
// ===== library types =====

// folder: LStream/DataTypes

TYPE "LStream_typeElement"
TITLE = LStream_typeElement
// describes the element for LStream libraries, by providing key-value pair and the depth of the element
   STRUCT
      "type" : SInt := -1;   // Type of element XML/JSON; -1 = inital value; 0 = Element/Object; 1 = Attribute/Array; 2 = Text/String; 3 = Number; 4 = Boolean / Type of element; -1 = inital value; 0 = Element/Object; 1 = Attribute/Array; 2 = Text
      key : String;   // Key name of element
      value : String := 'NULL';   // Value of element, null key has no value
      depth : SInt := -1;   // Depth of the key nesting
   END_STRUCT;
END_TYPE

// folder: LStream

FUNCTION_BLOCK "LStream_JsonDeserializer"   // FB3, SCL
TITLE = LStream_JsonDeserializer / LStream_JsonParser
{ S7_Optimized_Access := 'TRUE' }
AUTHOR : DI_FA_S_SUP_EuC
FAMILY : LStream
VERSION : 1.0
// parses a JSON string provided in the raw paramter  and rebuilds the coinatend bytes into a tree structure / Parses JSON file, with or without seach option
   VAR_INPUT
      execute : Bool;   // Rising edge starts action once
      search : Bool;   // TRUE: Search option is acticve
   END_VAR
   VAR_OUTPUT
      done : Bool;   // TRUE: Commanded functionality has been completed successfully
      busy : Bool;   // TRUE: FB is not finished and new output values can be expected
      error : Bool;   // TRUE: An error occurred during the execution of the FB
      status : Word := 16#7000;   // 16#0000 - 16#7FFF: Status of the FB, 16#8000 - 16#FFFF: Error identification
      resultCount : Int;   // Count of parsed JSON elements
   END_VAR
   VAR_IN_OUT
      tree : Array[*] of "LStream_typeElement";   // JSON tree containing the stored data
      raw : Array[*] of Byte;   // raw JSON data to parse in byte format
   END_VAR
   VAR
      statExecuteOld : Bool;   // Old value of 'execute' input for edge detection
      statDone : Bool;   // Static value for output 'done'
      statBusy : Bool;   // Static value for output 'busy'
      statError : Bool;   // Static value for output 'error'
      statStatus : Word := 16#7000;   // Static value for output 'status'
      statFBState : DInt := 0;   // State in the state machine of the FB
      statCountOfTree : Int;   // Static count of tree fields
      statCountOfRaw : Int;   // Static count of raw fields
      statResultCount : Int;   // Static value of result count
      statRawIndex : Int;   // Static value of raw index
      instWatchdog : IEC_TIMER;   // instance of watchdog timer
      statSearch : Bool;   // TRUE: Only keys provided in tree will be parsed
      statKeyValueFound : Bool;   // TRUE: Key exisits in raw data
      statTreeIndex : Int;   // Static value of tree index
      statSearchIndex : DInt;   // Static search
      statDepth : SInt := -1;   // Static value of JSON depth
      statOpen : Bool;   // TRUE: Key or Value is opened
      statInfoStartIndex : Int;   // Start index of current info in raw key or value
      statIgnorableCharacter : Bool;   // Next character to be ignored
      statInfoLen : UInt;   // Current information length key or value
      statKey : String;   // Static key string
      statValue : String;   // Static value string
      statKeyNotFoundCount : Int;   // Count of provided keys that weren't found
      statArrayOpen : Bool;   // TRUE: New JSON array is open
      statObjectArray : Bool;   // TRUE: Is type array of obejct
      statType : SInt;   // Current type of element
      statDefineValueType : Bool;   // TRUE: Value Type can be defined
      statArrayName : String;   // Name of array
   END_VAR
   VAR_TEMP
      tempExecute : Bool;   // Temporary value for input 'execute'
      tempRawIndex : Int;   // Index of raw field
      tempKeyToFind : String;   // Provided key to which the value should be found
      tempSearchResult : DInt;   // Temp value of search result
   END_VAR
   VAR CONSTANT
      FB_STATE_NO_PROCESSING : DInt := 0;   // FB state: No processing
      FB_STATE_PARSE : DInt := 1;   // FB state: Processing Parsing
      STATUS_EXECUTION_FINISHED : Word := 16#0000;   // Execution finished without errors
      STATUS_NO_CALL : Word := 16#7000;   // No job being currently processed
      STATUS_FIRST_CALL : Word := 16#7001;   // First call after incoming new job (rising edge 'execute')
      STATUS_SUBSEQUENT_CALL : Word := 16#7002;   // Subsequent call during active processing without further details
      ERR_TREE_ARRAY_TOO_SMALL : Word := 16#8201;   // Error: provided array to too small
      ERR_EMPTY_RAW_DATA : Word := 16#8401;   // Error: no raw data provided
      ERR_UNDEFINED_STATE : Word := 16#8600;   // Error: due to an undefined state in state machine
      JSON_QUTATIONMARK : Byte := 16#22;   // ASCII code for '"'
      JSON_COLON : Byte := 16#3A;   // ASCII code for ':'
      JSON_COMMA : Byte := 16#2C;   // ASCII code for ','
      JSON_BRACES_OPEN : Byte := 16#7B;   // ASCII code for '{'
      JSON_BRACES_CLOSE : Byte := 16#7D;   // ASCII code for '}'
      JSON_BRACKETS_OPEN : Byte := 16#5B;   // ASCII code for '['
      JSON_BRACKETS_CLOSE : Byte := 16#5D;   // ASCII code for ]
      "JSON_PROTECTION_KEY_\" : Byte := 16#5C;   // ASCII coder for / indicates closing / ASCII coder for \ indicates closing
      "JSON_CLOSE_KEY_/" : Byte := 16#2F;   // ASCII coder for / indicates closing
      LINE_FEED : Byte := 16#0A;   // ASCII code for line feed
      TAB : Byte := 16#09;   // ASCII code for TAB
      CARRIAGE_RETURN : Byte := 16#0D;   // ASCII code for carriage return
      SPACE : Byte := 16#20;   // ASCII code for blank space
      FIRST_DIM : USInt := 1;   // Constant for first array dimension
      MAX_LOOP_TIME : Time := T#3ms;   // Max duration of loop, will be continued in next cycle
      INVALID_SEARCH : DInt := -1;   // Return value if Search in LParse_FindStringInCharrArrayAdv was not successfull
      KEY_NOT_FOUND : String := 'Key not found';   // Value string in case key wasn't found
      INCREMENT_BY_ONE : USInt := 1;   // Constant to increment by one
      DECREMENT_BY_ONE : SInt := 1;   // Constant to decrement by one
      DECREMENT_BY_TWO : SInt := 2;   // Constant to decrement by one / Constant to decrement by two
      OBJECT : SInt := 0;   // Constant for value typ object / Constant for typ object
      "ARRAY" : SInt := 1;   // Constant for value typ array / Constant for typ array
      "STRING" : SInt := 2;   // Constant for value type string
      NUMBER : SInt := 3;   // Constant for value type number
      BOOLEAN : SInt := 4;   // Constant for value type boolean
      DEPTH_NOT_DEFINED : Int := -1;   // Constant indicating depth wasn't yet defined
   END_VAR
BEGIN
   REGION BLOCK INFO HEADER
     //===============================================================================
     // SIEMENS AG / (c)Copyright 2021
     //-------------------------------------------------------------------------------
     // Title:            LStream_JsonDeserializer
     // Comment/Function: parses a JSON string provided in the raw paramter
     //                   and rebuilds the coinatend bytes into a tree structure
     // Library/Family:   LStream
     // Author:           DI FA S SUP E&C
     // Tested with:      S7-1500 V2.8
     // Engineering:      TIA Portal V16
     // Restrictions:     -- 
     // Requirements:     LStream_FindStringInByteArrayAdv(FC), LStream_typeElement(UDT)
     //-------------------------------------------------------------------------------
     // Change log table:
     // Version  | Date       | Expert in charge       | Changes applied
     //----------|------------|------------------------|------------------------------
     // 01.0.0 | 2021-03-10 | DI FA S SUP E&C          | First released version
     // 01.0.8 | 2021-09-23 | DI FA S SUP E&C          | Adjustment type definition & bug fixes
     //===============================================================================
   END_REGION

   #tempExecute := #execute; // Work with temporary value / create process image

   REGION TRIGGERING
     IF (#tempExecute = TRUE) AND (#statExecuteOld = FALSE) // Check if FB is triggered
       AND (#statStatus = #STATUS_NO_CALL)
     THEN // First call; initialize FB
       #statDone := FALSE;
       #statBusy := TRUE;
       #statError := FALSE;
       #statStatus := #STATUS_FIRST_CALL;
       // State machine - start processing
       #statFBState := #FB_STATE_PARSE;

       // Initialize functionality: reset of variables, diagnostics, etc.
       #statSearch := #search;
       #statCountOfRaw := DINT_TO_INT(UPPER_BOUND(ARR := #raw, DIM := #FIRST_DIM));
       #statCountOfTree := DINT_TO_INT(UPPER_BOUND(ARR := #tree, DIM := #FIRST_DIM));
       #statOpen := FALSE;
       #statDepth := -1;
       #statRawIndex := 0;
       #statTreeIndex := 0;
       #statInfoLen := 0;
       #statSearchIndex := 0;
       #statKeyNotFoundCount := 0;
       #statType := -1;
       #statDefineValueType := FALSE;
       #statObjectArray := FALSE;

     ELSIF (#statStatus = #STATUS_FIRST_CALL) THEN
       #statStatus := #STATUS_SUBSEQUENT_CALL;
     END_IF;

     // Edge detection 'execute' input
     #statExecuteOld := #tempExecute;
   END_REGION TRIGGERING

   IF (#statStatus = #STATUS_NO_CALL) THEN // Nothing to do -> End here to reduce "system load"
     RETURN;
   END_IF;

   REGION STATE_MACHINE

     CASE #statFBState OF // State machine of FB
       #FB_STATE_NO_PROCESSING:
         REGION NO PROCESSING
           // No processing active (Note: this state must always be present and left empty)
           ;
         END_REGION NO PROCESSING

       #FB_STATE_PARSE: // Processing active
         REGION PARSING

           //rest watchdog
           #instWatchdog.TON(IN := FALSE,
                             PT := #MAX_LOOP_TIME);
           //start watchdog
           #instWatchdog.TON(IN := TRUE,
                             PT := #MAX_LOOP_TIME);

           FOR #tempRawIndex := #statRawIndex TO #statCountOfRaw DO

             REGION FIND KEY
               //pre check if key exist in raw data, if search option is active
               IF (#statSearch AND #statKeyValueFound = FALSE) THEN
                 IF (#statTreeIndex < #statCountOfTree) THEN
                   #tempSearchResult := "LStream_FindStringInByteCharArrayAdv"(searchFor := #tree[#statTreeIndex].key, startPosition := #statSearchIndex, searchIn := #raw);
                   IF (#tempSearchResult = #INVALID_SEARCH) THEN
                     //case key not found
                     #tree[#statTreeIndex].value := #KEY_NOT_FOUND;
                     #statTreeIndex += #INCREMENT_BY_ONE;
                     #statKeyNotFoundCount += #INCREMENT_BY_ONE;
                   ELSE//case key found
                     //move read pointer to last found index
                     #statSearchIndex := #tempSearchResult;
                     #statKeyValueFound := TRUE;
                   END_IF;
                 END_IF;
               END_IF;
             END_REGION FIND KEY   


             CASE #raw[#tempRawIndex] OF

               #JSON_BRACES_OPEN:
                 REGION OBJECT OPEN     

                   #statDepth += USINT_TO_SINT(#INCREMENT_BY_ONE);
                   IF (#statDefineValueType) THEN
                     #statDefineValueType := FALSE;
                     #statType := #OBJECT;
                     #tree[#statTreeIndex - #DECREMENT_BY_ONE].type := #statType;
                   END_IF;
                 END_REGION OBJECT OPEN

               #JSON_BRACES_CLOSE:
                 REGION OBJECT CLOSE      

                   #statDepth -= #DECREMENT_BY_ONE;
                   //last element closed, and there is still info in the buffer, then write value to last key
                   IF (#statDepth = -1 AND #statInfoLen > 0) THEN
                     //in case of 0 length, Chars_To_Strig returns the maxium possible char combination
                     Chars_TO_Strg(Chars := #raw,
                                   pChars := #statInfoStartIndex,
                                   Cnt := #statInfoLen,
                                   Strg => #statValue);
                     #statInfoLen := 0;

                     //value Type wasn't yet definied must be either number or boolean
                     IF (#statDefineValueType) THEN
                       #statDefineValueType := FALSE;

                       IF #statValue = 'FALSE' OR #statValue = 'TRUE'
                         OR #statValue = 'false' OR #statValue = 'true' THEN
                         #statType := #BOOLEAN;
                       ELSE
                         #statType := #NUMBER;
                       END_IF;

                     END_IF;

                     IF (#statSearch) THEN

                       IF (#statTreeIndex > 0) THEN
                         //in case of 0 length, Chars_To_Strig returns the maxium possible char combination
                         IF (#statKey = #tree[#statTreeIndex - #DECREMENT_BY_ONE].key) THEN
                           //only write into tree, if key matches, otherwise continue with search for matching key
                           #tree[#statTreeIndex - #DECREMENT_BY_ONE].value := #statValue;
                           #tree[#statTreeIndex - #DECREMENT_BY_ONE].type := #statType;
                           #statKeyValueFound := FALSE;
                         END_IF;
                       ELSE 
                         IF (#statKey = #tree[#statTreeIndex].key) THEN
                           #tree[#statTreeIndex].value := #statValue;
                           #tree[#statTreeIndex].type := #statType;
                           #statKeyValueFound := FALSE;
                         END_IF;
                       END_IF;

                     ELSE // IF #search option isn't active (parse all) add key TO the current #tree index
                       #tree[#statTreeIndex - #DECREMENT_BY_ONE].value := #statValue;
                       #tree[#statTreeIndex - #DECREMENT_BY_ONE].type := #statType;
                     END_IF;
                   END_IF;
                 END_REGION OBJECT CLOSE

               #JSON_BRACKETS_OPEN:
                 REGION ARRAY OPEN

                   #statDepth += USINT_TO_SINT(#INCREMENT_BY_ONE);

                   IF (#statTreeIndex > 0) THEN
                     //
                     #tree[#statTreeIndex - #DECREMENT_BY_ONE].type := #ARRAY;

                     //save arrayName
                     #statArrayName := #tree[#statTreeIndex - #DECREMENT_BY_ONE].key;

                     #statTreeIndex += #INCREMENT_BY_ONE;

                   ELSE // first element, is of type array
                     #tree[#statTreeIndex].type := #ARRAY;
                   END_IF;

                   #statArrayOpen := TRUE;
                   #statObjectArray := FALSE;
                 END_REGION ARRAY OPEN

               #JSON_BRACKETS_CLOSE:
                 REGION ARRAY CLOSE
                   #statDepth -= #DECREMENT_BY_ONE;
                   #statArrayOpen := FALSE;

                 END_REGION ARRAY CLOSE

               #JSON_QUTATIONMARK:
                 REGION QUTATIONMARK
                   IF (#statOpen) THEN
                     IF (NOT (#raw[#tempRawIndex - #DECREMENT_BY_ONE] = #"JSON_PROTECTION_KEY_\")) THEN
                       // previous sign \ then allowed in string adjust
                       #statOpen := FALSE;
                     ELSE
                       #statInfoLen += #INCREMENT_BY_ONE;
                     END_IF;
                   ELSE
                     #statInfoStartIndex := #tempRawIndex + #INCREMENT_BY_ONE; //set reader to next sign
                     #statOpen := TRUE;
                     #statIgnorableCharacter := FALSE;
                     //Qutation mark after colomn indicates value is of type string
                     IF #statDefineValueType THEN
                       #statType := #STRING;
                       #tree[#statTreeIndex - #DECREMENT_BY_ONE].type := #statType;
                       #statDefineValueType := FALSE;
                     END_IF;

                   END_IF;
                 END_REGION QUTATIONMARK

               #JSON_COLON:
                 REGION COLON

                   //array is open, and a sperate key is found indication for array of objects
                   //
                   IF #statArrayOpen AND NOT #statObjectArray THEN
                     #statObjectArray := TRUE;
                     #statTreeIndex -= #DECREMENT_BY_ONE;
                   END_IF;

                   //error handling
                   IF (#statTreeIndex > #statCountOfTree) THEN
                     //data does not fit in the provided tree 
                     #statStatus := #ERR_TREE_ARRAY_TOO_SMALL;
                     #statDone := TRUE;
                     EXIT;
                   END_IF;

                   //write key, if colon is part of a string
                   IF (NOT #statOpen) THEN
                     Chars_TO_Strg(Chars := #raw,
                                   pChars := #statInfoStartIndex,
                                   Cnt := #statInfoLen,
                                   Strg => #statKey);
                     #statInfoLen := 0;

                     //After key was written, type of value can be definied, value can be object, array, string, number, or boolean
                     #statDefineValueType := TRUE;

                     IF (#statSearch) THEN
                       //only write into tree, if key matches, otherwise continue with search for matching key
                       IF (#statKey = #tree[#statTreeIndex].key) THEN
                         //#tree[#statTreeIndex].type := #statType;
                         #tree[#statTreeIndex].depth := #statDepth;
                         #statTreeIndex += #INCREMENT_BY_ONE;
                       END_IF;

                     ELSE// if search option isn't active (parse all) the add key to the current tree index 
                       #tree[#statTreeIndex].key := #statKey;
                       //#tree[#statTreeIndex].type := #statType;
                       #tree[#statTreeIndex].depth := #statDepth;
                       #tree[#statTreeIndex].value := 'NULL';
                       #statTreeIndex += #INCREMENT_BY_ONE;
                     END_IF;

                     #statInfoStartIndex := #tempRawIndex+1;

                   ELSE//case : included in string
                     #statInfoLen += #INCREMENT_BY_ONE;
                   END_IF;
                 END_REGION COLON

               #JSON_COMMA:
                 REGION COMMA

                   //error handling
                   IF (#statTreeIndex > #statCountOfTree + #INCREMENT_BY_ONE) THEN
                     //data does not fit in the provided tree 
                     #statStatus := #ERR_TREE_ARRAY_TOO_SMALL;
                     #statDone := TRUE;
                     EXIT;
                   END_IF;

                   IF (NOT #statOpen) THEN
                     //write value comma isn't part of string
                     IF (#statInfoLen > 0) THEN
                       //in case of 0 length, Chars_To_Strig returns the maxium possible char combination
                       Chars_TO_Strg(Chars := #raw,
                                     pChars := #statInfoStartIndex,
                                     Cnt := #statInfoLen,
                                     Strg => #statValue);
                       #statInfoLen := 0;
                     ELSE
                       #statValue := 'NULL';
                       #statDefineValueType := FALSE;
                       //no value Type deafult value type NULL/Default is correct
                     END_IF;

                     //value Type wasn't yet definied must be either number or boolean
                     IF (#statDefineValueType) THEN
                       #statDefineValueType := FALSE;

                       IF #statValue = 'FALSE' OR #statValue = 'TRUE'
                         OR #statValue = 'false' OR #statValue = 'true' THEN
                         #statType := #BOOLEAN;
                       ELSE
                         #statType := #NUMBER;
                       END_IF;

                     END_IF;
                     //add value always to the last JSON element
                     IF (#statSearch) THEN

                       IF (#statTreeIndex > 0) THEN
                         //in case of 0 length, Chars_To_Strig returns the maxium possible char combination
                         IF (#statKey = #tree[#statTreeIndex - #DECREMENT_BY_ONE].key) THEN
                           //only write into tree, if key matches, otherwise continue with search for matching key
                           #tree[#statTreeIndex - #DECREMENT_BY_ONE].value := #statValue;
                           #tree[#statTreeIndex].type := #statType;
                           #statKeyValueFound := FALSE;
                         END_IF;
                       ELSE
                         IF (#statKey = #tree[#statTreeIndex].key) THEN
                           // if search option isn't active (parse all) the add key to the current tree index 
                           #tree[#statTreeIndex].value := #statValue;
                           #tree[#statTreeIndex].type := #statType;
                           #statKeyValueFound := FALSE;
                         END_IF;
                       END_IF;

                     ELSE//search option isn't active
                       #tree[#statTreeIndex - #DECREMENT_BY_ONE].value := #statValue;
                       #tree[#statTreeIndex - #DECREMENT_BY_ONE].type := #statType;
                       //case simple array last information
                       IF (#tree[#statTreeIndex - #DECREMENT_BY_ONE].depth = #DEPTH_NOT_DEFINED) THEN
                         #tree[#statTreeIndex - #DECREMENT_BY_ONE].depth := #tree[#statTreeIndex - #DECREMENT_BY_TWO].depth;
                         #tree[#statTreeIndex - #DECREMENT_BY_ONE].key := #statArrayName;
                         //always take depth from previous entry of simple array e.g "ArrayName":["ArrayValue1","ArrayValue2"]
                       END_IF;
                     END_IF;

                     IF (#statArrayOpen AND NOT #statObjectArray) THEN
                       //only write if Array is open and simple array
                       //
                       #tree[#statTreeIndex- #DECREMENT_BY_ONE].key := #statArrayName;
                       #tree[#statTreeIndex - #DECREMENT_BY_ONE].depth := #statDepth;//#tree[#statTreeIndex - #DECREMENT_BY_TWO].depth +1;
                       #tree[#statTreeIndex- #DECREMENT_BY_ONE].type := #statType;
                       //always take depth from previous entry of simple array e.g "ArrayName":["ArrayValue1","ArrayValue2"]


                       // #tree[#statTreeIndex].key := #tree[#statTreeIndex - #DECREMENT_BY_ONE].key;
                       // #tree[#statTreeIndex].depth := #tree[#statTreeIndex - #DECREMENT_BY_ONE].depth;
                       // #tree[#statTreeIndex].type := #tree[#statTreeIndex - #DECREMENT_BY_ONE].type;
                       #statTreeIndex += #INCREMENT_BY_ONE;
                     END_IF;

                     #statInfoStartIndex := #tempRawIndex;

                   ELSE//case ; included in string
                     #statInfoLen += #INCREMENT_BY_ONE;
                   END_IF;
                 END_REGION

               #TAB, #LINE_FEED, #CARRIAGE_RETURN, #SPACE:
                 REGION READ TAB LINE FEED CARRIAGE RETURN   
                   IF (NOT #statOpen) THEN
                     //do nothing when tab, line feed, or carriage return
                     #statIgnorableCharacter := TRUE;
                   ELSE//case space included in string
                     #statInfoLen += #INCREMENT_BY_ONE;
                   END_IF;

                 END_REGION READ TAB LINE FEED CARRIAGE RETURN     


               ELSE // all other characters
                 REGION ALL OTHER SIGNS
                 IF (#statIgnorableCharacter = TRUE) THEN
                   #statIgnorableCharacter := FALSE;
                   #statInfoStartIndex := #tempRawIndex; // set KeyIndex after all ignorableCharacters are read
                   #statInfoLen += #INCREMENT_BY_ONE;
                 ELSE
                   #statInfoLen += #INCREMENT_BY_ONE;
                 END_IF;
                 END_REGION ALL OTHER SIGNS 
             END_CASE;

             #statRawIndex := #tempRawIndex;

             //quit and resume in next cycle if watchdogtimer is exceed
             IF (#instWatchdog.Q) THEN
               #statRawIndex += #INCREMENT_BY_ONE;
               EXIT;
             END_IF;

           END_FOR;

           //if parser is through the entire raw data or end of tree array reached
           IF (#statRawIndex >= #statCountOfRaw) OR (#statTreeIndex > #statCountOfTree) THEN
             #statStatus := #STATUS_EXECUTION_FINISHED;
             #statResultCount := #statTreeIndex - #statKeyNotFoundCount;
           END_IF;
         END_REGION PARSING

       ELSE // Undefined state in state machine reached
         REGION UNDEFINED STATE
           #statStatus := #ERR_UNDEFINED_STATE;
         END_REGION UNDEFINED STATE
     END_CASE;
   END_REGION STATE_MACHINE

   REGION OUTPUTS
     // Write outputs
     IF (#statStatus = #STATUS_EXECUTION_FINISHED) AND (#statDone = FALSE) THEN // Execution finished without errors
       REGION EXECUTION FINSIHED
         #statDone := TRUE;
         #statBusy := FALSE;
         #statError := FALSE;
         // execution aborted --> set state no processing
         #statFBState := #FB_STATE_NO_PROCESSING;
       END_REGION EXECUTION FINSIHED

     ELSIF (#statStatus.%X15 = TRUE) AND (#statError = FALSE) THEN // Error occurred (#statStatus is 16#8000 to 16#FFFF)
       REGION ERROR OCCURD
         #statDone := FALSE;
         #statBusy := FALSE;
         #statError := TRUE;
         // execution aborted --> set state no processing
         #statFBState := #FB_STATE_NO_PROCESSING;
       END_REGION ERROR OCCURD

     ELSIF (#tempExecute = FALSE) AND ((#statDone = TRUE) OR (#statError = TRUE)) THEN // Reset outputs
       REGION EXECUTE RESETED
         #statDone := FALSE;
         #statBusy := FALSE;
         #statError := FALSE;
         #statStatus := #STATUS_NO_CALL;
         // Reset application specific outputs
         #statResultCount := 0;
       END_REGION EXECUTE RESETED
     END_IF;

     REGION WRITE STATIC VALUES TO OUTPUTS
       #done := #statDone;
       #busy := #statBusy;
       #error := #statError;
       #status := #statStatus;

       ENO := TRUE;
       // Write application specific static values to outputs
       #resultCount := #statResultCount;
     END_REGION WRITE STATIC VALUES TO OUTPUT
   END_REGION OUTPUTS
END_FUNCTION_BLOCK

FUNCTION_BLOCK "LStream_XmlDeserializer"   // FB4, SCL
TITLE = LStream_XmlDeserializer / LStream_Xml
{ S7_Optimized_Access := 'TRUE' }
AUTHOR : DI_FA_S_SUP_EuC
FAMILY : LStream
VERSION : 1.0
// parses a XML string provided in the Raw parameter and rebuilds the contained tree structure / Function Block parses entire or partial XML into DB
   VAR_INPUT
      execute : Bool;   // Rising edge starts action once
      search : Bool;   // TRUE: Searches rawdata for the value of the provided treekeys
   END_VAR
   VAR_OUTPUT
      done : Bool;   // TRUE: Commanded functionality has been completed successfully
      busy : Bool;   // TRUE: FB is not finished and new output values can be expected
      error : Bool;   // TRUE: An error occurred during the execution of the FB
      status : Word := 16#7000;   // 16#0000 - 16#7FFF: Status of the FB, 16#8000 - 16#FFFF: Error identification
      resultCount : Int;   // Count of parsed XML elements
   END_VAR
   VAR_IN_OUT
      tree : Array[*] of "LStream_typeElement";   // Tree parsed information is written to, if search option active, keys must be provided
      raw : Array[*] of Byte;   // Byte array of raw xml data
   END_VAR
   VAR
      statOldExecute : Bool;   // Old value of 'execute' input for edge detection
      statDepth : SInt := -1;   // Static value of xml depth
      statError : Bool;   // Static value of error
      statBusy : Bool;   // Static value of busy
      statStatus : Word := 16#7000;   // Static value of status
      statFBState : USInt := 0;   // Static value of fb state
      statDone : Bool;   // Static value of done
      statResultCount : Int;   // Static value of result count
      instWatchdog : IEC_TIMER;   // Instance of watchdog timer
      statRawIndex : Int;   // Static value of raw index
      statTreeIndex : Int;   // Static value of tree index
      statCountOfTree : Int;   // Static count of tree fields
      statCountOfRaw : Int;   // Static count of raw fields
      statIsIgnorable : Bool;   // Ignore any sign
      statIsKeyOpen : Bool;   // TRUE: key is open, internal flag
      statIsValueOpen : Bool;   // TRUE: value is open, internal flag
      statInfoLen : UInt;   // Current information length key or value
      statLastElementTreeIndex : Int;   // Treeindex of last element found
      statIgnorableCharacter : Bool;   // Next character to be ignored
      statInfoStartIndex : Int;   // Start index of current info in raw key or value
      statKeyWritten : Bool;   // TRUE: key was written into tree
      statKey : String;   // Static key string
      statValue : String;   // Static value string
      statSearch : Bool;   // TRUE: Only keys provided in tree will be parsed
      statKeyFound : Bool;   // TRUE: Key exisits in raw data
      statKeyNotFoundCount : Int;   // Count of provided keys that weren't found
      statSearchIndex : DInt;   // Static search index
   END_VAR
   VAR_TEMP
      tempRawIndex : Int;   // Index of raw field
      tempExecute : Bool;   // Temp of input execute
      tempKeyToFind : String;   // Provided key to which the value should be found
      tempSearchResult : DInt;   // Temp value of search result
   END_VAR
   VAR CONSTANT
      INCREMENT_BY_ONE : SInt := 1;   // Constant to increment by one
      DECREMENT_BY_ONE : SInt := 1;   // Constant to decrement by one
      FB_STATE_NO_PROCESSING : USInt := 0;   // FB state no processing, ideal state
      FB_STATE_PARSE : USInt := 10;   // FB state parse xml
      FB_STATE_DONE : USInt := 70;   // FB state done
      STATUS_EXECUTION_FINISHED : Word := 16#0000;   // NO error - execution finished without errors
      STATUS_NO_CALL : Word := 16#7000;   // No job being currently processed
      STATUS_FIRST_CALL : Word := 16#7001;   // First call after incoming new job (rising edge 'execute')
      STATUS_SUBSEQUENT_CALL : Word := 16#7002;   // Subsequent call during active processing without further details
      ERR_TREE_ARRAY_TOO_SMALL : Word := 16#8201;   // Error: provided array to too small
      ERR_EMPTY_RAW_DATA : Word := 16#8401;   // Error: no raw data provided
      ERR_UNDEFINED_STATE : Word := 16#8600;   // Error: due to an undefined state in state machine
      XML_HEADER : Byte := 16#3F;   // ASCII code for ? indicates xml header
      XML_COMMENT : Byte := 16#21;   // ASCII code for ! indicates comment
      XML_ATTRIBUTE_OPEN : Byte := 16#22;   // ASCII code for " frames value
      XML_OPEN_KEY : Byte := 16#3C;   // ASCII code for < indicates a new key
      XML_WRITE_KEY_EQUALS : Byte := 16#3D;   // ASCII code for '=' indicates key is finished follows by value
      XML_WRITE_KEY_GREATER : Byte := 16#3E;   // ASCII code for > indicates key can be written
      XML_WRITE_KEY_SPACE : Byte := 16#20;   // ASCII codefor SPACE indicates key is finished
      XML_CLOSE_KEY_SLASH : Byte := 16#2F;   // ASCII code for / indicates closing
      CARRIAGE_RETURN : Byte := 16#0D;   // ASCII code for carriage return
      LINE_FEED : Byte := 16#0A;   // ASCII code for line feed
      TAB : Byte := 16#09;   // ASCII code for TAB
      EMPTY : SInt := 0;   // Constant for zero value
      ELEMENT : SInt := 0;   // Numerical identifier for XML type elemt
      ATTRIBUTE : SInt := 1;   // Numerical identifier for XML type attirbute
      TEXT : SInt := 2;   // Numerical identifier for XML type text
      FIRST_DIM : USInt := 1;   // Constant for first array dimension
      MAX_LOOP_TIME : Time := T#3ms;   // Max duration of loop, will be continued in next cycle
      INVALID_SEARCH : DInt := -1;   // Return value if Search in LParse_FindStringInCharrArrayAdv was not successfull
      KEY_NOT_FOUND : String := 'Key not found';   // String value in case key wasn't found
   END_VAR
BEGIN
   REGION BLOCK INFO HEADER
     //===============================================================================
     // SIEMENS AG / (c)Copyright 2021
     //-------------------------------------------------------------------------------
     // Title:            LStream_XmlDeserializer
     // Comment/Function: parses a XML string provided in the Raw parameter
     //                   and rebuilds the contained tree structure
     // Library/Family:   LStream
     // Author:           DI FA S SUP E&C
     // Tested with:      S7-1500 V2.8
     // Engineering:      TIA Portal V16
     // Restrictions:     --
     // Requirements:     LStream_FindStringInByteArrayAdv(FC), LStream_typeElement(UDT)
     //-------------------------------------------------------------------------------
     // Change log table:
     // Version  | Date       | Expert in charge | Changes applied
     //----------|------------|------------------|------------------------------------
     // 01.00.00 | 2021-03-10 | DI FA S SUP E&C  | First released version
     //===============================================================================
   END_REGION

   #tempExecute := #execute;

   REGION TRIGGERING 

     IF (#tempExecute = TRUE) AND (#statOldExecute = FALSE)
       AND (#statStatus = #STATUS_NO_CALL)
     THEN // First call; initialize FB

       #statDone := FALSE;
       #statBusy := TRUE;
       #statStatus := #STATUS_FIRST_CALL;

       // Initialize functionality: reset of variables, diagnostics, etc.
       #statSearch := #search;
       #statCountOfRaw := DINT_TO_INT(UPPER_BOUND(ARR := #raw, DIM := #FIRST_DIM));
       #statCountOfTree := DINT_TO_INT(UPPER_BOUND(ARR := #tree, DIM := #FIRST_DIM));
       #statDepth := 0;
       #statRawIndex := 0;
       #statTreeIndex := 0;
       #statIsIgnorable := FALSE;
       #statIsKeyOpen := FALSE;
       #statIsValueOpen := FALSE;
       #statKeyWritten := FALSE;
       #statInfoLen := 0;
       #statLastElementTreeIndex := 0;
       #statIgnorableCharacter := FALSE;
       #statInfoStartIndex := 0;
       #statKey := '';
       #statValue := '';
       #statKeyFound := FALSE;
       #statSearchIndex := 0;
       #statKeyNotFoundCount := 0;

       // State machine - start processing
       #statFBState := #FB_STATE_PARSE;

       IF (NOT (#statCountOfRaw > #EMPTY)) THEN
         #statStatus := #ERR_EMPTY_RAW_DATA;
       END_IF;

     ELSIF (#statStatus = #STATUS_FIRST_CALL) THEN
       #statStatus := #STATUS_SUBSEQUENT_CALL;

     END_IF;

     // Edge detection 'execute' input
     #statOldExecute := #tempExecute;
   END_REGION TRIGGERING 

   IF (#statStatus = #STATUS_NO_CALL) THEN // Nothing to do -> End here to reduce "system load"
     RETURN;
   END_IF;

   REGION PROGRAM LOGIC

     CASE #statFBState OF // State machine of FB

       #FB_STATE_NO_PROCESSING:
         REGION NO PROCESSING
           // No processing active (Note: this state must always be present AND left empty)
           ;
         END_REGION NO PROCESSING           

       #FB_STATE_PARSE:
         REGION PARSE XML

           //rest and start watchdog here so that for loop runs for a maximum of 5 seconds
           #instWatchdog.TON(IN := FALSE,
                             PT := #MAX_LOOP_TIME);
           //start watchdog
           #instWatchdog.TON(IN := TRUE,
                             PT := #MAX_LOOP_TIME);

           FOR #tempRawIndex := #statRawIndex TO #statCountOfRaw DO

             //pre check if key exist in raw data, only if search option is active and key wasn't already found
             IF (#statSearch AND #statKeyFound = FALSE) THEN
               IF (#statTreeIndex < #statCountOfTree) THEN
                 #tempSearchResult := "LStream_FindStringInByteCharArrayAdv"(searchFor := #tree[#statTreeIndex].key, startPosition := #statSearchIndex, searchIn := #raw);

                 IF (#tempSearchResult = #INVALID_SEARCH) THEN
                   //case key not found
                   #tree[#statTreeIndex].value := #KEY_NOT_FOUND;
                   #statTreeIndex += #INCREMENT_BY_ONE;
                   #statKeyNotFoundCount += #INCREMENT_BY_ONE;

                 ELSE //case key found
                   //move read pointer to last found index
                   #statSearchIndex := #tempSearchResult;
                   #statKeyFound := TRUE;
                 END_IF;
               END_IF;
             END_IF;

             //swich case of current byte
             CASE #raw[#tempRawIndex] OF

               #XML_OPEN_KEY:
                 REGION READ OPENING KEY SYMBOLS                            
                   //check if is XML Header or comment by looking ahead by one 
                   IF (#raw[#tempRawIndex + 1] = #XML_HEADER) OR (#raw[#tempRawIndex + 1] = #XML_COMMENT) THEN
                     //in xml case <? and <!, ignore all signs until header or comment is finished
                     #statIsIgnorable := true;
                     #statInfoLen := 0;
                     //rest length buffer

                     //look ahead for closing  
                   ELSIF (#raw[#tempRawIndex + 1] = #XML_CLOSE_KEY_SLASH) THEN
                     // xml case </ indicates closeing
                     #statIsKeyOpen := false;
                     #statInfoLen := 0;

                   ELSE //indicates opening 
                     IF (#statTreeIndex > #statCountOfTree + #INCREMENT_BY_ONE) THEN
                       //data does not fit in the provided tree
                       #statStatus := #ERR_TREE_ARRAY_TOO_SMALL;
                       #statDone := TRUE;
                       EXIT;
                     END_IF;

                     IF (#statInfoLen > #EMPTY AND #statIsKeyOpen = TRUE) THEN
                       //xml case >text< 

                       Chars_TO_Strg(Chars := #raw,
                                     pChars := #statInfoStartIndex,
                                     Cnt := #statInfoLen,
                                     Strg => #statValue);

                       //add value to the last xml element
                       IF (#statSearch) THEN // search option is active

                         //only write value into tree, if key matches, otherwise continue with search for matching key
                         IF (#statKey = #tree[#statTreeIndex - #DECREMENT_BY_ONE].key) THEN

                           #tree[#statTreeIndex - #DECREMENT_BY_ONE].depth := #statDepth;
                           #tree[#statTreeIndex - #DECREMENT_BY_ONE].value := #statValue;
                           #tree[#statTreeIndex - #DECREMENT_BY_ONE].type := #TEXT;

                         END_IF;

                       ELSE // if search option isn't active (parse all) the value must be attached to the last key
                         #tree[#statTreeIndex - #DECREMENT_BY_ONE].depth := #statDepth;
                         #tree[#statTreeIndex - #DECREMENT_BY_ONE].value := #statValue;
                         #tree[#statTreeIndex - #DECREMENT_BY_ONE].type := #TEXT;
                       END_IF;
                     END_IF;

                     // new element
                     #statKeyWritten := FALSE;
                     #statIsKeyOpen := TRUE;
                     #statDepth += #INCREMENT_BY_ONE;
                     #statInfoStartIndex := #tempRawIndex + #INCREMENT_BY_ONE;
                     #statInfoLen := 0;

                   END_IF;

                 END_REGION READ OPENING KEY SYMBOLS       

               #XML_WRITE_KEY_GREATER, #XML_WRITE_KEY_EQUALS, #XML_WRITE_KEY_SPACE:
                 REGION READ WRITING KEY SYMBOLS

                   IF (#statIsIgnorable = FALSE) THEN
                     IF (#statInfoLen > #EMPTY AND #statIsKeyOpen = TRUE) THEN

                       IF (#statTreeIndex > #statCountOfTree) THEN
                         //data does not fit in the provided tree
                         #statStatus := #ERR_TREE_ARRAY_TOO_SMALL;
                         #statDone := TRUE;
                         EXIT;
                       END_IF;

                       Chars_TO_Strg(Chars := #raw,
                                     pChars := #statInfoStartIndex,
                                     Cnt := #statInfoLen,
                                     Strg => #statKey);


                       IF (#statSearch) THEN
                         //only write into tree, if key matches, otherwise continue with search for matching key
                         IF (#statKey = #tree[#statTreeIndex].key) THEN
                           #tree[#statTreeIndex].depth := #statDepth;
                           #tree[#statTreeIndex].type := #ELEMENT;
                           #statTreeIndex += #INCREMENT_BY_ONE;
                           #statKeyFound := FALSE;
                         END_IF;

                       ELSE// if search option isn't active (parse all) the add key to the current tree index
                         #tree[#statTreeIndex].key := #statKey;
                         #tree[#statTreeIndex].type := #ELEMENT;
                         #tree[#statTreeIndex].depth := #statDepth;
                         #tree[#statTreeIndex].value := 'NULL';
                         #statLastElementTreeIndex := #statTreeIndex;
                         #statTreeIndex += #INCREMENT_BY_ONE;
                         #statKeyFound := FALSE;
                         #statKeyWritten := TRUE;

                       END_IF;

                       #statInfoLen := 0;

                     END_IF;

                     #statInfoStartIndex := #tempRawIndex + #INCREMENT_BY_ONE;

                   ELSIF (#statIsIgnorable = TRUE AND #raw[#tempRawIndex] = #XML_WRITE_KEY_GREATER) THEN
                     //xml case closing of <? and <!, stop ignoring all signs
                     //only if sign is >
                     #statIsIgnorable := FALSE;

                   END_IF;
                 END_REGION READ WRITING KEY SYMBOLS

               #XML_CLOSE_KEY_SLASH:
                 REGION READ DELIMETER /
                   #statDepth -= #DECREMENT_BY_ONE;
                   #statIsKeyOpen := false;

                   IF (#statTreeIndex > #statCountOfTree) THEN
                     //data does not fit in the provided tree
                     #statStatus := #ERR_TREE_ARRAY_TOO_SMALL;
                     #statDone := TRUE;
                     EXIT;
                   END_IF;

                   IF (#statKeyWritten = FALSE) THEN
                     Chars_TO_Strg(Chars := #raw,
                                   pChars := #statInfoStartIndex,
                                   Cnt := #statInfoLen,
                                   Strg => #statKey);

                     //only if key wasn't alrady written
                     IF (NOT (#tree[#statLastElementTreeIndex].key = #statKey)) THEN

                       IF (#statSearch) THEN
                         //only write into tree, if key matches, otherwise continue with search for matching key
                         IF (#statKey = #tree[#statTreeIndex].key) THEN
                           #tree[#statTreeIndex].depth := #statDepth;
                           #statLastElementTreeIndex := #statTreeIndex;
                           #statTreeIndex += #INCREMENT_BY_ONE;
                           #statKeyFound := FALSE;
                         END_IF;
                       ELSE
                         // if search option isn't active (parse all) the add key to the current tree index
                         #tree[#statTreeIndex].key := #statKey;
                         #tree[#statTreeIndex].type := #ELEMENT;
                         #tree[#statTreeIndex].depth := #statDepth;
                         #tree[#statTreeIndex].value := 'NULL';
                         #statLastElementTreeIndex := #statTreeIndex;
                         #statTreeIndex += #INCREMENT_BY_ONE;
                         #statKeyFound := FALSE;
                         #statKeyWritten := TRUE;
                         #statInfoStartIndex := #tempRawIndex + #INCREMENT_BY_ONE;
                       END_IF;
                     END_IF;

                     #statInfoLen := 0;
                   END_IF;

                 END_REGION READ DELIMETER /

               #XML_ATTRIBUTE_OPEN:
                 REGION READ VALUE SYMBOLES
                   IF (#statIsIgnorable = FALSE) THEN

                     IF (#statIsValueOpen = false) THEN //first enter indicates begin of value
                       #statIsValueOpen := true;
                       #statInfoStartIndex := #tempRawIndex + #INCREMENT_BY_ONE;

                     ELSE // second enter indicates end of value
                       #statIsValueOpen := false;

                       IF (#statTreeIndex > #statCountOfTree + #INCREMENT_BY_ONE) THEN
                         //data does not fit in the provided tree 
                         #statStatus := #ERR_TREE_ARRAY_TOO_SMALL;
                         #statDone := TRUE;
                         EXIT;
                       END_IF;

                       //attach value to last key node
                       Chars_TO_Strg(Chars := #raw,
                                     pChars := #statInfoStartIndex,
                                     Cnt := #statInfoLen,
                                     Strg => #statValue);

                       IF (#statSearch) THEN
                         //only write into tree, if key matches, otherwise continue with search for matching key
                         IF (#statKey = #tree[#statTreeIndex - #DECREMENT_BY_ONE].key) THEN
                           #tree[#statTreeIndex - #DECREMENT_BY_ONE].depth := #statDepth;
                           #tree[#statTreeIndex - #DECREMENT_BY_ONE].value := #statValue;
                           #tree[#statTreeIndex - #DECREMENT_BY_ONE].type := #ATTRIBUTE;

                         END_IF;
                       ELSE
                         // if search option isn't active (parse all) the add key to the current tree index
                         #tree[#statTreeIndex - #DECREMENT_BY_ONE].value := #statValue;
                         #tree[#statTreeIndex - #DECREMENT_BY_ONE].type := #ATTRIBUTE;
                         #tree[#statTreeIndex - #DECREMENT_BY_ONE].depth := #statDepth;

                         #statIsValueOpen := false;
                       END_IF;
                       #statInfoLen := 0;
                     END_IF;
                   END_IF;
                 END_REGION READ VALUE SYMBOLES     

               #TAB, #LINE_FEED, #CARRIAGE_RETURN:
                 REGION READ TAB LINE FEED CARRIAGE RETURN                      
                   #statIgnorableCharacter := TRUE;
                   //do nothing when tab, line feed, or carriage return
                 END_REGION READ TAB LINE FEED CARRIAGE RETURN

               ELSE//all other characters  
                 REGION READ OTHER SIGN
                   IF (#statIgnorableCharacter = TRUE) THEN
                     #statIgnorableCharacter := FALSE;
                     #statInfoStartIndex := #tempRawIndex; // set KeyIndex after all ignorableCharacters are read

                   END_IF;
                   //count length in case not header or comment
                   IF (#statIsIgnorable = FALSE) THEN
                     #statInfoLen += SINT_TO_UINT(#INCREMENT_BY_ONE);
                   END_IF;

                 END_REGION READ OTHER SIGN                         

             END_CASE;
             #statRawIndex := #tempRawIndex;

             //quit and resume in next cycle if watchdogtimer is exceed
             IF (#instWatchdog.Q) THEN
               #statRawIndex += #INCREMENT_BY_ONE;
               EXIT;
             END_IF;
           END_FOR;

           //if parser is through the entire raw data or end of tree array reached
           IF (#statRawIndex >= #statCountOfRaw) OR (#statTreeIndex > #statCountOfTree) THEN
             #statStatus := #STATUS_EXECUTION_FINISHED;
             #statResultCount := #statTreeIndex - #statKeyNotFoundCount;
           END_IF;
         END_REGION PARSE XML              

       ELSE // Undefined state in state machine reached
         REGION UNDEFINED STATE
           #statStatus := #ERR_UNDEFINED_STATE;
         END_REGION UNDEFINED STATE
     END_CASE;

   END_REGION PROGRAM LOGIC

   REGION OUTPUTS

     // Write outputs
     IF (#statStatus = #STATUS_EXECUTION_FINISHED) AND (#statDone = FALSE) THEN // Execution finished without errors
       REGION EXECUTION FINISHED
         #statDone := TRUE;
         #statBusy := FALSE;
         #statError := FALSE;
         // execution aborted --> set state no processing
         #statFBState := #FB_STATE_NO_PROCESSING;
       END_REGION EXECUTION FINISHED

     ELSIF (#statStatus.%X15 = TRUE) AND (#statError = FALSE) THEN // Error occurred (#statStatus is 16#8000 to 16#FFFF)
       REGION ERROR OCCURED
         #statDone := FALSE;
         #statBusy := FALSE;
         #statError := TRUE;
         // execution aborted --> set state no processing
         #statFBState := #FB_STATE_NO_PROCESSING;
       END_REGION ERROR OCCURED

     ELSIF (#tempExecute = FALSE) AND ((#statDone = TRUE) OR (#statError = TRUE)) THEN // Reset outputs
       REGION EXECUTE RESETED
         #statDone := FALSE;
         #statBusy := FALSE;
         #statError := FALSE;
         #statStatus := #STATUS_NO_CALL;
         // Reset application specific outputs
         #statResultCount := 0;
       END_REGION EXECUTE RESETED
     END_IF;

     REGION WRITE STATIC VALUES TO OUTPUTS
       // write application specific temp values to outputs
       #resultCount := #statResultCount;
       #done := #statDone;
       #error := #statStatus.%X15;
       #status := #statStatus;
       #busy := #statBusy;

     END_REGION WRITE STATIC VALUES TO OUTPUTS

   END_REGION OUTPUTS
END_FUNCTION_BLOCK

FUNCTION_BLOCK "LStream_JsonSerializer"   // FB5, SCL
TITLE = LStream_JsonDeserializer / LStream_JsonParser
{ S7_Optimized_Access := 'TRUE' }
AUTHOR : DI_FA_S_SUP_EuC
FAMILY : LStream
VERSION : 1.0
// parses a JSON string provided in the raw paramter  and rebuilds the coinatend bytes into a tree structure / Parses JSON file, with or without seach option
   VAR_INPUT
      execute : Bool;   // Rising edge starts action once
   END_VAR
   VAR_OUTPUT
      done : Bool;   // TRUE: Commanded functionality has been completed successfully
      busy : Bool;   // TRUE: FB is not finished and new output values can be expected
      error : Bool;   // TRUE: An error occurred during the execution of the FB
      status : Word := 16#7000;   // 16#0000 - 16#7FFF: Status of the FB, 16#8000 - 16#FFFF: Error identification
      count : UInt;   // Count of char/ byte info elements in byte array / Count of parsed JSON elements
   END_VAR
   VAR_IN_OUT
      tree : Array[*] of "LStream_typeElement";   // JSON tree containing the stored data
      jsonByteArray : Array[*] of Byte;   // JSON structure as array of bytes / raw JSON data to parse in byte format
   END_VAR
   VAR
      statExecuteOld : Bool := FALSE;   // Old value of 'execute' input for edge detection
      statDone : Bool := FALSE;   // Static value for output 'done'
      statBusy : Bool := FALSE;   // Static value for output 'busy'
      statError : Bool := FALSE;   // Static value for output 'error'
      statCount : UInt := 0;   // Static value for ouput 'count'
      statStatus : Word := 16#7000;   // Static value for output 'status'
      statFbState : DInt := 0;   // State in the state machine of the FB
      statFbPreviousState : DInt := 0;   // Previos state in the state machine of the FB
      statFbNextState : DInt := 0;   // Next state in the state machine of the FB
      statIndexJsonByteArray : UInt := 0;   // Index indicating current element of byte array to be written
      statIndexTreeArray : UInt := 0;   // Index indicating current element of tree array to be read
      statTreeLen : DInt := 0;   // Length of tree array
      statJsonByteLen : DInt := 0;   // Length of xml byte array / Length of json byte array
      statInfoToWrite : String := '';   // Static value of current information that should be written to XML
      statIsLastElement : Bool := FALSE;   // TRUE: is last element in tree array
      statLastElementIsClosed : Bool := FALSE;   // TRUE: Last JSON element is closed / TRUE: Last XML element is closed
      statStackIndexOpenElement : Array[0..#STACK_SIZE] of Char;   // Stack of open elements
      statStackIndex : Int := -1;   // Stack pointer and current depth / Stack pointer
      instWatchdog : IEC_TIMER;   // Instance for watchdog timer
      statIsArrayOpen : Bool;   // Static value indicating weather an array is open
      statIsArrayFieldClosed : Bool;   // Static value indicating weather an array field was closed
      statIsFirstElement : Bool;   // TRUE: first field of simple array
      statFirstArrayKey : String;   // First key of array, used to check for new array beginning
      statArrayName : String;   // Name of Array
   END_VAR
   VAR_TEMP
      tempExecute : Bool;   // Temporary value for input 'execute'
      tempCntCharsAdded : UInt;   // Temporary value indicating count of chars added to byte array
   END_VAR
   VAR CONSTANT
      FB_STATE_NO_PROCESSING : DInt := 0;   // FB state: No processing
      FB_STATE_NEXT_ELEMENT : DInt := 1;   // FB state: Get Next Element
      FB_STATE_VALUE_TYPE : DInt := 2;   // FB state: Switch Value type / FB state: Switch Element type
      FB_STATE_WRITE_TO_JSON : DInt := 3;   // FB state: Add Informationto xml byte array
      FB_STATE_CLOSE_STACK_ELEMENT : DInt := 4;   // FB state: Close Parent Element
      STATUS_EXECUTION_FINISHED : Word := 16#0000;   // Execution finished without errors
      STATUS_NO_CALL : Word := 16#7000;   // No job being currently processed
      STATUS_FIRST_CALL : Word := 16#7001;   // First call after incoming new job (rising edge 'execute')
      STATUS_SUBSEQUENT_CALL : Word := 16#7002;   // Subsequent call during active processing without further details
      ERR_UNDEFINED_STATE : Word := 16#8600;   // Error: due to an undefined state in state machine
      ERR_IN_BLOCK_OPERATION : Word := 16#8001;   // Error: wrong operation of the function block
      ERR_PARAMETRIZATION : Word := 16#8200;   // Error: during parameterization
      ERR_PROCESSING_EXTERN : Word := 16#8400;   // Error: when processing from outside (e. g. wrong I/O signals, axis not referenced)
      ERR_UNDEFINED_TYPE : Word := 16#8401;   // Error: user enter undefined type
      ERR_UNEXPECTED_DEPTH : Word := 16#8402;   // Error: provided json tree structure is too deep / Error: provided xml tree structure is too deep
      ERR_DEPTH_MISSING : Word := 16#8403;   // Error: provided json tree structure does not contain correct depth / Error: provided xml tree structure does not contain correct depth
      ERR_PROCESSING_INTERN : Word := 16#8600;   // Error: when processing internally (e. g. when calling a system function)
      ERR_TREE_OUT_OF_BOUNDS : Word := 16#8601;   // Error: tree array out of bounds
      ERR_JSON_OUT_OF_BOUNDS : Word := 16#8602;   // Error: byte array out of bounds
      ERR_STACK_OUT_OF_BOUNDS : Word := 16#8603;   // Error: stack array out of bounds
      ERR_AREA_RESERVED : Word := 16#8800;   // Error: reserved area
      ERR_USER_DEFINED_CLASSES : Word := 16#9000;   // Error: user-defined error classes
      QUTATIONMARK : Char := '"';   // ASCII code for '"'
      COLON : Char := ':';   // ASCII code for ':'
      COMMA : Char := ',';   // ASCII code for ','
      BRACES_OPEN : Char := '{';   // ASCII code for '{'
      BRACES_CLOSE : Char := '}';   // ASCII code for '}'
      BRACKETS_OPEN : Char := '[';   // ASCII code for '['
      BRACKETS_CLOSE : Char := ']';   // ASCII code for ]
      "PROTECTION_KEY_\" : Char := '\';   // ASCII coder for / indicates closing / ASCII coder for \ indicates closing
      LINE_FEED : Char := '$L';   // ASCII code for line feed
      TAB : Char := '$T';   // ASCII code for TAB
      CARRIAGE_RETURN : Char := '$R';   // ASCII code for carriage return
      SPACE : Char := ' ';   // ASCII code for blank space
      FIRST_DIM : USInt := 1;   // Constant for first array dimension
      MAX_REPEAT_TIME : Time := T#3ms;   // Max duration of loop, will be continued in next cycle
      INVALID_SEARCH : DInt := -1;   // Return value if Search in LParse_FindStringInCharrArrayAdv was not successfull
      KEY_NOT_FOUND : String := 'Key not found';   // Value string in case key wasn't found
      INCREMENT_BY_ONE : USInt := 1;   // Constant to increment by one
      DECREMENT_BY_ONE : SInt := 1;   // Constant to decrement by one
      OBJECT : SInt := 0;   // Constant for value typ object / Constant for typ object
      "ARRAY" : SInt := 1;   // Constant for value typ array / Constant for typ array
      "STRING" : SInt := 2;   // Constant for value type string
      NUMBER : SInt := 3;   // Constant for value type number
      BOOLEAN : SInt := 4;   // Constant for value type boolean
      NEXT_INDEX : UInt := 1;   // Constant value to get next index
      STACK_SIZE : UInt := 10;   // Constant for Stack Size, equals max depth
      WHITE_SPACE : Char := ' ';   // ASCII code for white space
      NOT_INITALYZED : SInt := -1;   // Constant value representing not initalyzed tree element
      EMPTY : String;   // Constant value representing an empty string
      NULL : String := 'NULL';   // Constant value representing null
   END_VAR
   // statStackIndexOpenElement[0] := '$00';
   // statStackIndexOpenElement[1] := '$00';
BEGIN
   REGION BLOCK INFO HEADER
     //===============================================================================
     // SIEMENS AG / (c)Copyright 2021
     //-------------------------------------------------------------------------------
     // Title:            LStream_JsonSerializer
     // Comment/Function: parses a JSON string provided in the raw paramter
     //                   and rebuilds the coinatend bytes into a tree structure
     // Library/Family:   LStream
     // Author:           DI FA S SUP E&C
     // Tested with:      S7-1500 V2.8
     // Engineering:      TIA Portal V16
     // Restrictions:     -- 
     // Requirements:     LStream_typeElement(UDT)
     //-------------------------------------------------------------------------------
     // Change log table:
     // Version  | Date       | Expert in charge       | Changes applied
     //----------|------------|------------------------|------------------------------
     // 01.00.00 | 2021-06-10 | DI FA S SUP E&C        | First released version
     //===============================================================================
   END_REGION

   #tempExecute := #execute; // Work with temporary value / create process image

   REGION TRIGGERING
     IF (#tempExecute = TRUE) AND (#statExecuteOld = FALSE) // Check if FB is triggered
       AND (#statStatus = #STATUS_NO_CALL)
     THEN // First call; initialize FB
       #statDone := FALSE;
       #statBusy := TRUE;
       #statError := FALSE;
       #statStatus := #STATUS_FIRST_CALL;
       // State machine - start processing
       #statFbState := #FB_STATE_NEXT_ELEMENT;

       //Initialize functionality: reset OF variables, diagnostics, etc.
       #statJsonByteLen := UPPER_BOUND(ARR := #jsonByteArray, DIM := #FIRST_DIM);
       #statTreeLen := UPPER_BOUND(ARR := #tree, DIM := #FIRST_DIM);
       #statIndexTreeArray := 0;
       #statIndexJsonByteArray := 0;
       #statIsLastElement := FALSE;
       #statLastElementIsClosed := FALSE;
       #statStackIndex := -1;
       #statIsArrayOpen := FALSE;

     ELSIF (#statStatus = #STATUS_FIRST_CALL) THEN
       #statStatus := #STATUS_SUBSEQUENT_CALL;
     END_IF;

     // Edge detection 'execute' input
     #statExecuteOld := #tempExecute;
   END_REGION TRIGGERING

   IF (#statStatus = #STATUS_NO_CALL) THEN // Nothing to do -> End here to reduce "system load"
     RETURN;
   END_IF;

   REGION STATE_MACHINE

     //rest and start watchdog here so that repeat until has a maximum duration of constant MAX_LOOP_TIME
     #instWatchdog.TON(IN := FALSE,
                       PT := #MAX_REPEAT_TIME);
     //start watchdog
     #instWatchdog.TON(IN := TRUE,
                       PT := #MAX_REPEAT_TIME);
     REPEAT
       #statFbPreviousState := #statFbState;

       CASE #statFbState OF // State machine of FB

         #FB_STATE_NO_PROCESSING:
           REGION NO PROCESSING
             // No processing active (Note: this state must always be present and left empty)
             ;
           END_REGION NO PROCESSING

         #FB_STATE_NEXT_ELEMENT: // Work on next Element
           REGION NEXT_ELEMENT
             REGION ERROR HANDLING
               //check for last Element, either end of provided tree reached, or tree element is -1 = not initalized
               //this prevents index out of bounds error
               IF (#statIndexTreeArray = #statTreeLen - 1) OR #tree[#statIndexTreeArray + #NEXT_INDEX].type = #NOT_INITALYZED THEN
                 #statIsLastElement := TRUE;

               ELSIF (#statIndexTreeArray = #statTreeLen) THEN
                 //Error: Tree out of Bound
                 #statStatus := #ERR_TREE_OUT_OF_BOUNDS;
               END_IF;

               //Error: provided XML tree is too deep
               //max depth size allowed is size of stack, otherwise array out of bounds error will occur
               IF (#tree[#statIndexTreeArray].depth = #STACK_SIZE) THEN
                 #statStatus := #ERR_UNEXPECTED_DEPTH;
               ELSIF (#tree[#statIndexTreeArray].depth = #NOT_INITALYZED) THEN
                 //depth wasn't provided by user
                 #statStatus := #ERR_DEPTH_MISSING;
               END_IF;
             END_REGION #ERROR_HANDLING

             //must only be set once, reset after every new element
             #statIsFirstElement := FALSE;
             // stackIndex is used as current depth, is initalized wih -1 therefore first element, will always open an object 
             IF #statStackIndex < 0 THEN
               //open object
               #statInfoToWrite := CONCAT(IN1 := CHAR_TO_STRING(#BRACES_OPEN), IN2 := CHAR_TO_STRING(#WHITE_SPACE));
               //increase stack index and push closing elements on to it
               #statStackIndex += #INCREMENT_BY_ONE;
               #statStackIndexOpenElement[#statStackIndex] := #BRACES_CLOSE;
             END_IF;

             //in case Array is open, save the first key of the first field.
             //This is later used to check when new array field beginn 
             IF (#statIsArrayOpen AND #statFirstArrayKey = '') THEN

               //prevent that simple #ARRAY structure e.g "ArrayName":["ArrayValue1","ArrayValue2"]
               //is misread as key is array name that field info
               IF #statArrayName <> #tree[#statIndexTreeArray].key THEN
                 #statFirstArrayKey := #tree[#statIndexTreeArray].key;
               // ELSE //simple array case

               //   IF NOT #statIsFirstElement AND NOT #statIsSecondElement THEN
               //     //set flag that it is simple array
               //     //array field so no uneccarsy comma is written
               //     //as now depth change occurs
               //     #statIsFirstElement := TRUE;
               //   ELSE
               //     #statIsFirstElement := FALSE;
               //     #statIsSecondElement := TRUE;
               //   END_IF;
               END_IF;

               //in case Array is open, and current key matches first key of the first field,
               //indication of new array field, append open symbolic
             ELSIF (#statIsArrayOpen AND #statFirstArrayKey = #tree[#statIndexTreeArray].key) THEN

               IF NOT #statIsArrayFieldClosed THEN
                 //field wasn't close as no deeper hierarchy exist, therfore the normal close opeartion is invalid
                 //close now here
                 #statInfoToWrite := CONCAT(IN1 := CHAR_TO_STRING(#BRACES_CLOSE), IN2 := CHAR_TO_STRING(#COMMA));
                 #statStackIndex -= #DECREMENT_BY_ONE;
               ELSE //reset flag
                 #statIsArrayFieldClosed := FALSE;
               END_IF;
               //open object
               #statInfoToWrite := CONCAT(IN1 := #statInfoToWrite, IN2 := CHAR_TO_STRING(#BRACES_OPEN), IN3 := CHAR_TO_STRING(#WHITE_SPACE));
               //increase stack index and push closing elements on to it
               #statStackIndex += #INCREMENT_BY_ONE;
               #statStackIndexOpenElement[#statStackIndex] := #BRACES_CLOSE;
             END_IF;

             IF NOT (#statIsArrayOpen AND #statArrayName = #tree[#statIndexTreeArray].key)  THEN
               //write key not in case array is open and key is the same array name
               //this indicates simple array structure e.g "ArrayName":["ArrayValue1","ArrayValue2"]
               //write key -> "key":
               #statInfoToWrite := CONCAT(IN1 := #statInfoToWrite, IN2 := CHAR_TO_STRING(#QUTATIONMARK),
                                          IN3 := #tree[#statIndexTreeArray].key, IN4 := CHAR_TO_STRING(#QUTATIONMARK),
                                          IN5 := CHAR_TO_STRING(#COLON), IN6 := CHAR_TO_STRING(#WHITE_SPACE));

             END_IF;

             //Move to state Write
             #statFbState := #FB_STATE_WRITE_TO_JSON;
             //Set state, that should be executed after writing
             //move on to next state
             #statFbNextState := #FB_STATE_VALUE_TYPE;

           END_REGION NEXT_ELEMENT 

         #FB_STATE_VALUE_TYPE: // Depending on value type, write value
           REGION VALUE DEPENDECY OF TYPE
             CASE #tree[#statIndexTreeArray].type OF

               #OBJECT:
                 REGION OBJECT
                   //nothing to do when type is object just add line feed, { openning will occur with next depth
                   #statInfoToWrite := CONCAT(IN1 := #statInfoToWrite, IN2 := CHAR_TO_STRING(#BRACES_OPEN));
                   //increase stack index and push closing elements on to it
                   #statStackIndex += #INCREMENT_BY_ONE;
                   #statStackIndexOpenElement[#statStackIndex] := #BRACES_CLOSE;
                 END_REGION OBJECT

               #ARRAY:
                 REGION ARRAY

                   IF (NOT #statIsArrayOpen) THEN
                     #statIsFirstElement := TRUE;
                     #statIsArrayOpen := TRUE;
                     //set Name of Array
                     #statArrayName := #tree[#statIndexTreeArray].key;

                     #statInfoToWrite := CONCAT(IN1 := CHAR_TO_STRING(#BRACKETS_OPEN), IN2 := CHAR_TO_STRING(#WHITE_SPACE));
                     //increase stack index and push closing elements on to it
                     #statStackIndex += #INCREMENT_BY_ONE;
                     #statStackIndexOpenElement[#statStackIndex] := #BRACKETS_CLOSE;

                     //case for underlaying object structure in array, prevent depth of simple array to have leading {
                     //simple array always has arrayname as key
                     IF #tree[#statIndexTreeArray].depth < #tree[#statIndexTreeArray + #NEXT_INDEX].depth
                       AND #tree[#statIndexTreeArray+ #NEXT_INDEX].key <> #statArrayName THEN
                       //open object
                       #statInfoToWrite := CONCAT(IN1 := #statInfoToWrite, IN2 := CHAR_TO_STRING(#BRACES_OPEN));
                       //increase stack index and push closing elements on to it
                       #statStackIndex += #INCREMENT_BY_ONE;
                       #statStackIndexOpenElement[#statStackIndex] := #BRACES_CLOSE;
                     END_IF;

                   END_IF;

                   // //null indicating that it is array definition, array information is written sepe
                   // //otherwise write value as string - value enclosed with quotation mark 
                   // IF(#tree[#statIndexTreeArray].value <> #NULL) THEN
                   //   #statInfoToWrite := CONCAT(IN1 := #statInfoToWrite, IN2 := CHAR_TO_STRING(#QUTATIONMARK),
                   //                              IN3 := #tree[#statIndexTreeArray].value, IN4 := CHAR_TO_STRING(#QUTATIONMARK));
                   // END_IF;
                 END_REGION ARRAY 

               #STRING:
                 REGION STRING

                   //wirte value as string - value enclosed with quotation mark 
                   IF (#tree[#statIndexTreeArray].value <> #NULL) THEN
                     #statInfoToWrite := CONCAT(IN1 := #statInfoToWrite, IN2 := CHAR_TO_STRING(#QUTATIONMARK),
                                                IN3 := #tree[#statIndexTreeArray].value, IN4 := CHAR_TO_STRING(#QUTATIONMARK));

                   ELSE // empty value still needs "" otherwise syntax error
                     #statInfoToWrite := CONCAT(IN1 := #statInfoToWrite, IN2 := CHAR_TO_STRING(#QUTATIONMARK),
                                                IN3 := CHAR_TO_STRING(#QUTATIONMARK));
                   END_IF;
                 END_REGION STRING

               #NUMBER, #BOOLEAN:
                 REGION NUMBER_BOOLEAN
                   //wirte value as number or boolean - value enclosed without quotation mark 
                   IF (#tree[#statIndexTreeArray].value <> #NULL) THEN
                     #statInfoToWrite := CONCAT(IN1 := #statInfoToWrite,
                                                IN2 := #tree[#statIndexTreeArray].value);
                   END_IF;
                 END_REGION NUMBER_BOOLEAN

               ELSE // Undefined state in state machine reached
                 REGION UNDEFINED STATE
                   #statStatus := #ERR_UNDEFINED_STATE;
                 END_REGION UNDEFINED STATE          

             END_CASE;

             //Move to state Write
             #statFbState := #FB_STATE_WRITE_TO_JSON;

             //Set state, that should be executed after writing
             //move on to next state
             #statFbNextState := #FB_STATE_NEXT_ELEMENT;

             IF #statIsLastElement OR #tree[#statIndexTreeArray].depth > #tree[#statIndexTreeArray + #NEXT_INDEX].depth THEN
               //Next Element has lower depth, therefore Elements have to be closed
               #statFbNextState := #FB_STATE_CLOSE_STACK_ELEMENT;
             ELSIF #statIsLastElement OR #tree[#statIndexTreeArray].depth = #tree[#statIndexTreeArray + #NEXT_INDEX].depth AND  NOT #statIsFirstElement THEN
                #statInfoToWrite := CONCAT(IN1 := #statInfoToWrite,
                                           IN2 := CHAR_TO_STRING(#COMMA));
             END_IF;
             //#statInfoToWrite := CONCAT(IN1 := #statInfoToWrite, IN2 := CHAR_TO_STRING(#LINE_FEED));



             //increase tree index to access next element 
             #statIndexTreeArray += #INCREMENT_BY_ONE;

           END_REGION VALUE DEPENDECY OF TYPE

         #FB_STATE_WRITE_TO_JSON: // Write to Byte Array
           REGION WRITE TO JSON                
             //add information to json byte array
             IF ((INT_TO_UINT(LEN(#statInfoToWrite)) + #statIndexJsonByteArray) < #statJsonByteLen) THEN
               Strg_TO_Chars(Strg := #statInfoToWrite,
                             pChars := #statIndexJsonByteArray,
                             Cnt => #tempCntCharsAdded,
                             Chars := #jsonByteArray);


               #statInfoToWrite := #EMPTY;
               //move index of byte array 
               #statIndexJsonByteArray += #tempCntCharsAdded;
               //move to next state previously allocated
               #statFbState := #statFbNextState;
             ELSE // Error: Index out of bounds
               #statStatus := #ERR_JSON_OUT_OF_BOUNDS;
             END_IF;

             IF #statLastElementIsClosed THEN
               //writer has written last information and execution is done
               #statStatus := #STATUS_EXECUTION_FINISHED;
               //current index equals count/size of json byte array
               #statCount := #statIndexJsonByteArray;
             END_IF;
           END_REGION WRITE TO JSON

         #FB_STATE_CLOSE_STACK_ELEMENT: //Close Open Stack Elements
           REGION CLOSE ELEMENT FROM STACK
             //close element with syntax </key>

             IF #statStackIndex >= 0 THEN //more open elements available, not all elements are closed

               //statInfoToWrite --> } or ]
               #statInfoToWrite := CHAR_TO_STRING(#statStackIndexOpenElement[#statStackIndex]);

               IF #statInfoToWrite = #BRACKETS_CLOSE THEN
                 //reset flag
                 #statIsArrayOpen := FALSE;

                 //first array key is used to recognize,
                 //beginning of new array field reset here, so it can be check for emptiness
                 #statFirstArrayKey := '';
               END_IF;

               //pop element from stack 
               #statStackIndex -= SINT_TO_INT(#DECREMENT_BY_ONE);

               IF #statStackIndex >= 0 THEN //more open elements available, not all elements are closed
                 //look at current stack item depth, if next tree element has 
                 IF NOT #statIsLastElement AND #statStackIndex = #tree[#statIndexTreeArray].depth THEN
                   //move to next element
                   //write comma as JSON dictates same depth a divided by comma,
                   //here we move on to the next elment with the same depth
                   #statInfoToWrite := CONCAT(IN1:=  #statInfoToWrite, IN2:= CHAR_TO_STRING(#COMMA));

                   // //if Array is still open and the same lenght is reached,
                   // //new element in array, distinguish new entry with BRACES
                   IF #statIsArrayOpen THEN
                     #statInfoToWrite := CONCAT(IN1 := #statInfoToWrite, IN2 := CHAR_TO_STRING(#BRACES_CLOSE), IN3 := CHAR_TO_STRING(#COMMA));
                     //pop element from stack 
                     #statStackIndex -= SINT_TO_INT(#DECREMENT_BY_ONE);
                     #statIsArrayFieldClosed := TRUE;
                   //   #statInfoToWrite := CONCAT(IN1 := #statInfoToWrite, IN2 := CHAR_TO_STRING(#BRACES_OPEN));
                   //   //increase stack index and push closing elements on to it
                   //   #statStackIndex += #INCREMENT_BY_ONE;
                   //   #statStackIndexOpenElement[#statStackIndex] := #BRACES_CLOSE;
                   END_IF;
                   #statFbNextState := #FB_STATE_NEXT_ELEMENT;

                 ELSE
                   //do nothing and return to fb state close element 
                   #statFbNextState := #FB_STATE_CLOSE_STACK_ELEMENT;
                 END_IF;

               ELSE
                 //no more open Elements, last Element was closed
                 #statIsLastElement := TRUE;

                 //only if this flag is set, can writer be finished
                 #statLastElementIsClosed := TRUE;

               END_IF;

             ELSE
               //no more open Elements, last Element was closed
               #statIsLastElement := TRUE;

               //only if this flag is set, can writer be finished
               #statLastElementIsClosed := TRUE;

             END_IF;
             //Move to state Write
             #statFbState := #FB_STATE_WRITE_TO_JSON;

           END_REGION CLOSE ELEMENT FROM STACK

         ELSE // Undefined state in state machine reached
           REGION UNDEFINED STATE
             #statStatus := #ERR_UNDEFINED_STATE;
           END_REGION UNDEFINED STATE     

       END_CASE;
       //Leave state machine if one of the following condition is true
       //1. state has not changed
       //2. error has occured
       //3. watchdog timer expired 
       //4. execution has finished
       // otherwise stay in state machine
     UNTIL (#statFbPreviousState = #statFbState OR #statStatus.%X15
       OR #instWatchdog.Q OR #statStatus = #STATUS_EXECUTION_FINISHED)
     END_REPEAT;
   END_REGION STATE_MACHINE

   REGION OUTPUTS
     // Write outputs
     IF (#statStatus = #STATUS_EXECUTION_FINISHED) AND (#statDone = FALSE) THEN // Execution finished without errors
       REGION EXECUTION FINSIHED
         #statDone := TRUE;
         #statBusy := FALSE;
         #statError := FALSE;
         // execution aborted --> set state no processing
         #statFbState := #FB_STATE_NO_PROCESSING;
       END_REGION EXECUTION FINSIHED

     ELSIF (#statStatus.%X15 = TRUE) AND (#statError = FALSE) THEN // Error occurred (#statStatus is 16#8000 to 16#FFFF)
       REGION ERROR OCCURED
         #statDone := FALSE;
         #statBusy := FALSE;
         #statError := TRUE;
         // execution aborted --> set state no processing
         #statFbState := #FB_STATE_NO_PROCESSING;
       END_REGION ERROR OCCURED

     ELSIF (#tempExecute = FALSE) AND ((#statDone = TRUE) OR (#statError = TRUE)) THEN // Reset outputs
       REGION EXECUTE RESETTED
         #statDone := FALSE;
         #statBusy := FALSE;
         #statError := FALSE;
         #statStatus := #STATUS_NO_CALL;
         // Reset application specific outputs
         #statCount := 0;
       END_REGION EXECUTE RESETTED
     END_IF;

     REGION WRITE STATIC VALUES TO OUTPUTS
       #done := #statDone;
       #busy := #statBusy;
       #error := #statError;
       #status := #statStatus;
       //  ENO mechanism is not used 
       ENO := TRUE;
       // Write application specific static values to outputs
       #count := #statCount;
     END_REGION WRITE STATIC VALUES TO OUTPUTS
   END_REGION OUTPUTS
END_FUNCTION_BLOCK

FUNCTION_BLOCK "LStream_XmlSerializer"   // FB13, SCL
TITLE = LStream_XmlSerializer / LStream_XmlWriter
{ S7_Optimized_Access := 'TRUE' }
AUTHOR : DI_FA_S_SUP_E&C
FAMILY : LStream
VERSION : 1.0
// FB converts prefilled array of udt LParse_typeElement to a xml structure.
// XML structure is returned as a byte array
// FB  converts prefilled array of udt LParse_typeElement to a xml structure.
// XML structure is returned as a byte array
   VAR_INPUT
      execute : Bool;   // Rising edge starts action once
   END_VAR
   VAR_OUTPUT
      done : Bool;   // TRUE: Commanded functionality has been completed successfully
      busy : Bool;   // TRUE: FB is not finished and new output values can be expected
      error : Bool;   // TRUE: An error occurred during the execution of the FB
      status : Word := 16#7000;   // 16#0000 - 16#7FFF: Status of the FB, 16#8000 - 16#FFFF: Error identification
      count : UInt;   // Count of char/ byte info elements in byte array
   END_VAR
   VAR_IN_OUT
      tree : Array[*] of "LStream_typeElement";
      xmlByteArray : Array[*] of Byte;   // XML structure as array of bytes
   END_VAR
   VAR
      statExecuteOld : Bool := FALSE;   // Old value of 'execute' input for edge detection
      statDone : Bool := FALSE;   // Static value for output 'done'
      statBusy : Bool := FALSE;   // Static value for output 'busy'
      statError : Bool := FALSE;   // Static value for output 'error'
      statCount : UInt := 0;   // Static value for ouput 'count'
      statStatus : Word := 16#7000;   // Static value for output 'status'
      statFbState : DInt := 0;   // State in the state machine of the FB
      statFbPreviousState : DInt := 0;   // Previos state in the state machine of the FB
      statFbNextState : DInt := 0;   // Next state in the state machine of the FB
      statIndexXmlByteArray : UInt := 0;   // Index indicating current element of byte array to be written
      statIndexTreeArray : UInt := 0;   // Index indicating current element of tree array to be read
      statTreeLen : DInt := 0;   // Length of tree array
      statXmlByteLen : DInt := 0;   // Length of xml byte array
      statInfoToWrite : String := '';   // Static value of current information that should be written to XML
      statIsLastElement : Bool := FALSE;   // TRUE: is last element in tree array
      statLastElementIsClosed : Bool := FALSE;   // TRUE: Last XML element is closed
      statStackIndexOpenElement : Array[0..#STACK_SIZE] of UInt;   // Stack of open elements
      statStackIndex : Int := -1;   // Stack pointer
      instWatchdog : IEC_TIMER;   // Instance for watchdog timer
   END_VAR
   VAR_TEMP
      tempExecute : Bool;   // Temporary value for input 'execute'
      tempCntCharsAdded : UInt;   // Temporary value indicating count of chars added to byte array
   END_VAR
   VAR CONSTANT
      FB_STATE_NO_PROCESSING : DInt := 0;   // FB state: No processing
      FB_STATE_XML_HEADER : DInt := 1;   // FB state: Write XML Header
      FB_STATE_NEXT_ELEMENT : DInt := 2;   // FB state: Get Next Element
      FB_STATE_ELEMENT_TYPE : DInt := 3;   // FB state: Switch Element type
      FB_STATE_WRITE_TO_XML : DInt := 4;   // FB state: Add Informationto xml byte array
      FB_STATE_CLOSE_STACK_ELEMENT : DInt := 5;   // FB state: Close Parent Element
      STATUS_EXECUTION_FINISHED : Word := 16#0000;   // Execution finished without errors
      STATUS_NO_CALL : Word := 16#7000;   // No job being currently processed
      STATUS_FIRST_CALL : Word := 16#7001;   // First call after incoming new job (rising edge 'execute')
      STATUS_SUBSEQUENT_CALL : Word := 16#7002;   // Subsequent call during active processing without further details
      ERR_UNDEFINED_STATE : Word := 16#8600;   // Error: due to an undefined state in state machine
      ERR_IN_BLOCK_OPERATION : Word := 16#8001;   // Error: wrong operation of the function block
      ERR_PARAMETRIZATION : Word := 16#8200;   // Error: during parameterization
      ERR_PROCESSING_EXTERN : Word := 16#8400;   // Error: when processing from outside (e. g. wrong I/O signals, axis not referenced)
      ERR_UNDEFINED_TYPE : Word := 16#8401;   // Error: user enter undefined type
      ERR_UNEXPECTED_DEPTH : Word := 16#8402;   // Error: provided xml tree structure is too deep
      ERR_DEPTH_MISSING : Word := 16#8403;   // Error: provided xml tree structure does not contain correct depth
      ERR_PROCESSING_INTERN : Word := 16#8600;   // Error: when processing internally (e. g. when calling a system function)
      ERR_TREE_OUT_OF_BOUNDS : Word := 16#8601;   // Error: tree array out of bounds
      ERR_XML_OUT_OF_BOUNDS : Word := 16#8602;   // Error: byte array out of bounds
      ERR_STACK_OUT_OF_BOUNDS : Word := 16#8603;   // Error: stack array out of bounds
      ERR_AREA_RESERVED : Word := 16#8800;   // Error: reserved area
      ERR_USER_DEFINED_CLASSES : Word := 16#9000;   // Error: user-defined error classes
      INCREMENT_BY_ONE : SInt := 1;   // Constant to increment by one
      DECREMENT_BY_ONE : SInt := 1;   // Constant to decrement by one
      ELEMENT : SInt := 0;   // Numerical identifier for XML type element
      ATTRIBUTE : SInt := 1;   // Numerical identifier for XML type attirbute
      TEXT : SInt := 2;   // Numerical identifier for XML type text
      FIRST_DIM : USInt := 1;   // Constant for first array dimension
      MAX_REPEAT_TIME : Time := T#3ms;   // Max duration of loop, will be continued in next cycle
      XML_HEADER : String := '<?xml version="1.0" encoding="UTF-8" ?>';   // XML Header, leads every XML File
      XML_KEY_OPEN : Char := '<';   // ASCII code for < indicates a new key
      XML_ATTRIBUTE_OPEN : String := '="';   // ASCII code for '=' indicates key is finished follows by value
      XML_KEY_CLOSE_GREATER : Char := '>';   // ASCII code for > indicates key can be written
      XML_KEY_CLOSE_SLASH : Char := '/';   // ASCII code for / indicates closing
      XML_ATTRIBUTE_CLOSE : Char := '"';   // ASCII code for " frames value
      NEXT_INDEX : UInt := 1;   // Constant value to get next index
      STACK_SIZE : UInt := 10;   // Constant for Stack Size, equals max depth
      WHITE_SPACE : Char := ' ';   // ASCII code for white space
      NOT_INITALYZED : SInt := -1;   // Constant value representing not initalyzed tree element
   END_VAR
   // statStackIndexOpenElement[0] := 0;
   // statStackIndexOpenElement[1] := 0;
BEGIN
   REGION BLOCK INFO HEADER
     //===============================================================================
     // SIEMENS AG / (c)Copyright 2021
     //-------------------------------------------------------------------------------
     // Title:            LStream_XmlSerializer
     // Comment/Function: FB converts prefilled array of udt LParse_typeElement to a xml structure.
     //                   XML structure is returned as a Byte array
     // Library/Family:   LStream
     // Author:           DI FA S SUP E&C 
     // Tested with:      S7-1500 V2.8
     // Engineering:      TIA Portal V16
     // Restrictions:     -
     // Requirements:     LStream_typeElement(UDT)
     //-------------------------------------------------------------------------------
     // Change log table:
     // Version  | Date       | Expert in charge       | Changes applied
     //----------|------------|------------------------|------------------------------
     // 01.00.00 | 2021-03-10 | DI FA S SUP E&C        | First released version
     //===============================================================================
   END_REGION

   #tempExecute := #execute; // Work with temporary value / create process image

   REGION TRIGGERING
     IF (#tempExecute = TRUE) AND (#statExecuteOld = FALSE) // Check if FB is triggered
       AND (#statStatus = #STATUS_NO_CALL)
     THEN // First call; initialize FB
       #statDone := FALSE;
       #statBusy := TRUE;
       #statError := FALSE;
       #statStatus := #STATUS_FIRST_CALL;
       // State machine - start processing
       #statFbState := #FB_STATE_XML_HEADER;

       //Initialize functionality: reset OF variables, diagnostics, etc.
       #statXmlByteLen := UPPER_BOUND(ARR := #xmlByteArray, DIM := #FIRST_DIM);
       #statTreeLen := UPPER_BOUND(ARR := #tree, DIM := #FIRST_DIM);
       #statIndexTreeArray := 0;
       #statIndexXmlByteArray := 0;
       #statIsLastElement := FALSE;
       #statLastElementIsClosed := FALSE;
       #statStackIndex := -1;

     ELSIF (#statStatus = #STATUS_FIRST_CALL) THEN
       #statStatus := #STATUS_SUBSEQUENT_CALL;
     END_IF;

     // Edge detection 'execute' input
     #statExecuteOld := #tempExecute;
   END_REGION TRIGGERING

   IF (#statStatus = #STATUS_NO_CALL) THEN // Nothing to do -> End here to reduce "system load"
     RETURN;
   END_IF;

   REGION STATE_MACHINE

     //rest and start watchdog here so that repeat until has a maximum duration of constant MAX_LOOP_TIME
     #instWatchdog.TON(IN := FALSE,
                       PT := #MAX_REPEAT_TIME);
     //start watchdog
     #instWatchdog.TON(IN := TRUE,
                       PT := #MAX_REPEAT_TIME);
     REPEAT
       #statFbPreviousState := #statFbState;

       CASE #statFbState OF // State machine of FB

         #FB_STATE_NO_PROCESSING:
           REGION NO PROCESSING
             // No processing active (Note: this state must always be present and left empty)
             ;
           END_REGION NO PROCESSING

         #FB_STATE_XML_HEADER: // Add xml Header 
           REGION WRITE XML HEADER
             // Write XML Header at the beginning of byte array
             #statInfoToWrite := #XML_HEADER;
             //Move to state Write
             #statFbState := #FB_STATE_WRITE_TO_XML;
             //Set state, that should be executed after writing
             #statFbNextState := #FB_STATE_NEXT_ELEMENT;
           END_REGION WRITE XML HEADER    

         #FB_STATE_NEXT_ELEMENT: // Get Next Element and write tree key
           REGION GET NEXT ELEMENT 

             //check for last Element, either end of provided tree reached, or tree element is -1 = not initalized
             //this prevents index out of bounds error
             IF (#statIndexTreeArray = #statTreeLen - 1) OR #tree[#statIndexTreeArray + #NEXT_INDEX].type = #NOT_INITALYZED THEN
               #statIsLastElement := TRUE;

             ELSIF (#statIndexTreeArray = #statTreeLen) THEN
               //Error: Tree out of Bound
               #statStatus := #ERR_TREE_OUT_OF_BOUNDS;
             END_IF;

             //Error: provided XML tree is too deep
             //max depth size allowed is size of stack, otherwise array out of bounds error will occur
             IF (#tree[#statIndexTreeArray].depth = #STACK_SIZE) THEN
               #statStatus := #ERR_UNEXPECTED_DEPTH;
             ELSIF (#tree[#statIndexTreeArray].depth = #NOT_INITALYZED) THEN
               #statStatus := #ERR_DEPTH_MISSING;
             END_IF;

             IF (#tree[#statIndexTreeArray].type <> #ATTRIBUTE) THEN
               //key is element or text set open element and add key
               //statInfoToWrite --> <key
               #statInfoToWrite := CONCAT(IN1 := CHAR_TO_STRING(#XML_KEY_OPEN),
                                          IN2 := #tree[#statIndexTreeArray].key);

               //add index number to stack, to access element from stack and close element
               IF (#statStackIndex < #STACK_SIZE) THEN
                 #statStackIndex += SINT_TO_INT(#INCREMENT_BY_ONE);
                 #statStackIndexOpenElement[#statStackIndex] := #statIndexTreeArray;

               ELSE //Error: Stack out of Bound
                 #statStatus := #ERR_STACK_OUT_OF_BOUNDS;
               END_IF;

             ELSE // tree field is attribute
               //key is attribute name,add key 
               //statInfoToWrite --> key
               #statInfoToWrite := #tree[#statIndexTreeArray].key;
             END_IF;

             //Move to state Write
             #statFbState := #FB_STATE_WRITE_TO_XML;
             //Set state, that should be executed after writing
             #statFbNextState := #FB_STATE_ELEMENT_TYPE;
           END_REGION GET NEXT ELEMENT

         #FB_STATE_ELEMENT_TYPE: // Check Type and write tree value
           REGION WRITE VALUE
             CASE #tree[#statIndexTreeArray].type OF

               #ATTRIBUTE:
                 REGION ATTRIBUTE
                   //ATTRIBUTE - Attribute name is udt tree[i].key, attribute value is tree[i].value

                   //create string for attribute syntax ="value" to be written in next step
                   //statInfoToWrite --> ="value"
                   #statInfoToWrite := CONCAT(IN1 := #XML_ATTRIBUTE_OPEN,
                                              IN2 := #tree[#statIndexTreeArray].value,
                                              IN3 := #XML_ATTRIBUTE_CLOSE);

                   IF (#statIsLastElement) THEN
                     //element can be closed, syntax />

                     //statInfoToWrite --> ="value"/>
                     #statInfoToWrite := CONCAT(IN1 := #statInfoToWrite,
                                                IN2 := #XML_KEY_CLOSE_SLASH,
                                                IN3 := #XML_KEY_CLOSE_GREATER);

                     //element was closed, pop index from stack, only open elements continue to stay on stack 
                     #statStackIndex -= SINT_TO_INT(#DECREMENT_BY_ONE);

                     //move on to stack and see if parent element can be closed as well, atleast root element still located on stack
                     #statFbNextState := #FB_STATE_CLOSE_STACK_ELEMENT;//set state to closing all open elements

                   ELSE//more information available, peek at next field, to define what the next stat should be
                     IF #tree[#statIndexTreeArray + #NEXT_INDEX].type = #ATTRIBUTE THEN
                       // Add space for syntax, in case more than one attribute in element
                       //next tree field is also attribute, keep Element open
                       //="value"' '
                       #statInfoToWrite := CONCAT(IN1 := #statInfoToWrite,
                                                  IN2 := #WHITE_SPACE);

                       #statFbNextState := #FB_STATE_NEXT_ELEMENT;

                       //increase tree index to access next element
                       #statIndexTreeArray += SINT_TO_UINT(#INCREMENT_BY_ONE);

                     ELSIF #tree[#statIndexTreeArray + #NEXT_INDEX].depth <= #tree[#statIndexTreeArray].depth THEN
                       //element can be closed, no child element, only sibiling or parent element, syntax />

                       //="value"/>
                       #statInfoToWrite := CONCAT(IN1 := #statInfoToWrite,
                                                  IN2 := #XML_KEY_CLOSE_SLASH,
                                                  IN3 := #XML_KEY_CLOSE_GREATER);

                       //element was closed, pop index from stack, only open elements continue to stay on stack 
                       #statStackIndex -= SINT_TO_INT(#DECREMENT_BY_ONE);

                       IF #tree[#statIndexTreeArray + #NEXT_INDEX].depth < #tree[#statIndexTreeArray].depth THEN
                         //next element is parent element, stack must be closed

                         //Set state, that should be executed after writing
                         #statFbNextState := #FB_STATE_CLOSE_STACK_ELEMENT;

                       ELSE
                         //next element is sibiling with same depth, parent element stays open, access next element
                         //Set state, that should be executed after writing
                         #statFbNextState := #FB_STATE_NEXT_ELEMENT;
                         //increase index 
                         #statIndexTreeArray += SINT_TO_UINT(#INCREMENT_BY_ONE);
                       END_IF;

                     ELSE // case next element depth > current depth, element has child element

                       //element can be closed with syntax >
                       //statInfoToWrite --> ="value">
                       #statInfoToWrite := CONCAT(IN1 := #statInfoToWrite,
                                                  IN2 := CHAR_TO_STRING(#XML_KEY_CLOSE_GREATER));

                       //Set state, that should be executed after writing
                       #statFbNextState := #FB_STATE_NEXT_ELEMENT;
                       //increase tree index to access next element
                       #statIndexTreeArray += SINT_TO_UINT(#INCREMENT_BY_ONE);
                     END_IF;
                   END_IF;
                 END_REGION ATTRIBUTE

               #TEXT:
                 REGION TEXT
                   //TEXT - Element name is tree[i]key, text value is tree[i].value

                   //create string for text syntax >"Text"<
                   //statInfoToWrite --> ="value">
                   #statInfoToWrite := CONCAT(IN1 := #XML_KEY_CLOSE_GREATER,
                                              IN2 := #tree[#statIndexTreeArray].value);
                   IF (#statIsLastElement) THEN
                     //Set state, that should be executed after writing
                     //move on to stack and see if parent element can be closed as well, at least current and root element still located on stack
                     #statFbNextState := #FB_STATE_CLOSE_STACK_ELEMENT;//set state to closing all

                   ELSE//more information available, peek at next field

                     IF #tree[#statIndexTreeArray + #NEXT_INDEX].depth > #tree[#statIndexTreeArray].depth THEN

                       //Set state, that should be executed after writing
                       #statFbNextState := #FB_STATE_NEXT_ELEMENT;
                       //increase tree index to access next element
                       #statIndexTreeArray += SINT_TO_UINT(#INCREMENT_BY_ONE);
                     ELSE
                       //close text element with syntax text</key>, 
                       //Set state, that should be executed after writing
                       #statFbNextState := #FB_STATE_CLOSE_STACK_ELEMENT;
                     END_IF;

                   END_IF;
                 END_REGION TEXT

               #ELEMENT:
                 REGION ELEMENT
                   //ELEMENT - Element name is tree[i]key, element has no value. value is null

                   IF #tree[#statIndexTreeArray].type = #ELEMENT
                     AND #tree[#statIndexTreeArray + 1].type = #ELEMENT //if next element is also of type elment and isn't a child element
                     AND #tree[#statIndexTreeArray + 1].depth <= #tree[#statIndexTreeArray].depth THEN

                     //element can be closed, syntax />
                     //statInfo to Write --> />
                     #statInfoToWrite := CONCAT(IN1 := #XML_KEY_CLOSE_SLASH,
                                                IN2 := #XML_KEY_CLOSE_GREATER);

                     //element was closed, pop index from stack, only open elements continue to stay on stack 
                     #statStackIndex -= SINT_TO_INT(#DECREMENT_BY_ONE);

                     IF (#statIsLastElement) THEN
                       //Set state, that should be executed after writing
                       #statFbNextState := #FB_STATE_CLOSE_STACK_ELEMENT;//set state to closing all

                     ELSE//more information available, peek at next field

                       IF (#tree[#statIndexTreeArray + #NEXT_INDEX].depth < #tree[#statIndexTreeArray].depth) THEN
                         //next element is parent element, stack must be closed
                         //Set state, that should be executed after writing
                         #statFbNextState := #FB_STATE_CLOSE_STACK_ELEMENT;
                       ELSE
                         //next Element is sibiling
                         //Set state, that should be executed after writing
                         #statFbNextState := #FB_STATE_NEXT_ELEMENT;
                         //increase tree index to access next element
                         #statIndexTreeArray += SINT_TO_UINT(#INCREMENT_BY_ONE);
                       END_IF;

                     END_IF;

                   ELSIF #tree[#statIndexTreeArray + #NEXT_INDEX].type = #ATTRIBUTE THEN
                     // when key is of type element, and next key is an attribite 
                     // 
                     // insert white space, otherwise xml syntax error <key attribitue
                     // statInfoToWrite --> WHITE_SPACE
                     #statInfoToWrite := #WHITE_SPACE;

                     //Set state, that should be executed after writing
                     #statFbNextState := #FB_STATE_NEXT_ELEMENT;
                     //increase tree index to access next element
                     #statIndexTreeArray += SINT_TO_UINT(#INCREMENT_BY_ONE);

                   ELSE// Child Element or last element

                     IF #statIsLastElement THEN
                       //element can be closed, syntax />
                       // statInfoToWrite --> />
                       #statInfoToWrite := CONCAT(IN1 := #XML_KEY_CLOSE_SLASH,
                                                  IN2 := #XML_KEY_CLOSE_GREATER);

